PROGRAM MAIN
VAR
	cnt			: UINT;
	
	fbLight00		: fbLightControl;
	fbLight01		: fbLightControl;
	fbLight02		: fbLightControl;
	fbLight03		: fbLightControl;
	fbLight04		: fbLightControl;
	fbLight05		: fbLightControl; // testje
	fbLight06		: fbLightControl;
	fbLight07		: fbLightControlV2;
	fbLight08		: fbLightControl_ButtonAndDetect;
	fbLight09		: fbLightControl;
	fbLight10		: fbLightControl;
	fbLight11		: fbLightControl;
	fbLight12		: fbLightControl;
	fbLight13		: fbLightControl;
	fbLight14		: fbLightControl;
//	fbLight15		: fbLightControl;
	
	bOutputActief	: BOOL;
	
	bForceOff		:BOOL;
	bForceOn		:BOOL;
	
	InputTriggerAllesUit		: R_trig; 
	
	LesruimteLichtAan: INT;
END_VAR

 cnt := cnt +1;



InputTriggerAllesUit(CLK := GVL.I_Input35 OR GVL.I_Input24 OR gvl.I_Input17);
	
// Actual light control

fbLight00(bButton:= GVL.I_Input32 , 
			bForceOff:= InputTriggerAllesUit.Q, 
			bForceOn:= , 
			bLight=> gvl.Q_Light07,
			bLight=> gvl.Q_Light04,
			);
// Grote WC hoofdlicht

GVL.Q_Light01 := GVL.I_Input09; //midden WC
GVL.Q_Light00 := GVL.I_Input13; // Grote WC 
GVL.Q_Light04 := GVL.I_Input10;// WC naast tech
GVL.Q_Light15 := GVL.I_Input14; // tech ruimte
GVL.Q_Light12 := GVL.I_Input08;// BergRuimte =Detector
GVL.Q_Light13 := GVL.I_Input11 OR GVL.I_Input12;// Gang deel2 detector


//verlichting Bureau
		


		

		
		// Licht Keuken
fbLight02(bButton:= GVL.I_Input03 OR GVL.I_Input23 ,  // check other button 
			bForceOff:= InputTriggerAllesUit.Q, 
			bForceOn:= , 
			bLight=> gvl.Q_Light02,
		);
		
// Licht Buiten	
fbLight03(bButton:= GVL.I_Input04 OR GVL.I_Input31 OR GVL.I_Input22, 
			bForceOff:= InputTriggerAllesUit.Q, 
			bForceOn:= , 
			bLight=> gvl.Q_Light03,
		);
		
// 	vergaderzaal

fbLight05(bButton:= GVL.I_Input21, 
			bForceOff:= InputTriggerAllesUit.Q, 
			bForceOn:= , 
			bLight=> gvl.Q_Light05
		);	
// Bureau

fbLight06(bButton:= GVL.I_Input01,
			bForceOff:= InputTriggerAllesUit.Q, 
			bForceOn:= , 
			
			bLight=> gvl.Q_Light06
		);	
// Lesruimte 	
fbLight07(bButtonhoofdFunctie:= GVL.I_Input02 OR GVL.I_Input15 ,
			bButton2 := GVL.I_Input18 OR GVL.I_Input16, // 16 should move to outside
			bForceOff:= InputTriggerAllesUit.Q, 
			bForceOn:= , 
			bLight1=> gvl.Q_Light07,
			bLight2=> gvl.Q_Light17
		);	
// Garage 	
fbLight08(bButton:= GVL.I_Input33 OR GVL.I_Input05 OR GVL.I_Input32 OR GVL.I_Input26,
			bDetection := GVL.I_Input37  ,
			bDeurDetectie :=  NOT(GVL.I_Input29) OR NOT(GVL.I_Input27),
			bForceOff:= InputTriggerAllesUit.Q, 
			bForceOn:= , 
			bInhibit:= InputTriggerAllesUit.Q, 
			bLight=> gvl.Q_Light08,
			bLight=> gvl.Q_Light09,
		);
// Deze knop laat toe om de detectie over te nemen 
// Logica nog te verbeteren met de alles uit samen te werken


(*TODO: remove after logic validation
gvl.Q_Light08 := gvl.Q_Light08 OR GVL.I_Input37;
gvl.Q_Light09 := gvl.Q_Light09 OR GVL.I_Input37;*)

// zaal boven
fbLight10(bButton:= GVL.I_Input34 OR GVL.I_Input06 OR GVL.I_Input25, 
			bForceOff:= InputTriggerAllesUit.Q, 
			bForceOn:= , 
			bLight=> gvl.Q_Light10,
			bLight=> gvl.Q_Light11
			);

// GrimeLicht Grote WC
fbLight14(bButton:= GVL.I_Input19 , 
			bForceOff:= InputTriggerAllesUit.Q, 
			bForceOn:= , 
			bLight=> gvl.Q_Light14
		);	

		
bOutputActief := fbLight00.bLight
				OR fbLight01.bLight
				OR fbLight02.bLight
				OR fbLight03.bLight
				OR fbLight04.bLight
				OR fbLight05.bLight
				OR fbLight06.bLight
				OR fbLight07.bLight1 OR fbLight07.bLight2
				OR fbLight08.bLight
				OR fbLight09.bLight
				OR fbLight10.bLight
				OR fbLight11.bLight
				OR fbLight12.bLight
				OR fbLight13.bLight
				OR fbLight14.bLight;

GVL.Q_Light16 :=  bOutputActief;				

// Activeer Verwarming

	GVL.LesruimteLichtAan := gvl.Q_Light07 OR gvl.Q_Light17 OR gvl.Q_Light02;
	GVL.BureauLichtAan	  := gvl.Q_Light06 ;
	GVL.Vergaderzaal	  := gvl.Q_Light05 ;

SturingVerwarming();

END_PROGRAM

(* stored: Version 1.1.0.1, ProductVersion 3.1.4024.12
   POU MAIN: Id {644e9ade-a57c-45cf-ab42-b4c8dbcedaa1}, SpecialFunc None *)
